FUNCTION_BLOCK TaskFB EXTENDS TaskBase
VAR_INPUT
END_VAR
VAR_OUTPUT
END_VAR
VAR
END_VAR

END_FUNCTION_BLOCK

(* stored: Version 1.1.0.1, ProductVersion 3.1.4024.12
   POU TaskFB: Id {8ce34e13-fd71-44c8-9783-8c2bb14c6857}, SpecialFunc None *)
